// TIA Portal V20 export
DATA_BLOCK "DB_Digital_Outputs"   // DB3
{ S7_Optimized_Access := 'TRUE' }
// stored: MemoryReserve 100
   VAR
      Digital_Output_0 : Bool;
      Digital_Output_1 : Bool;
      Digital_Output_2 : Bool;
      Digital_Output_3 : Bool;
      Digital_Output_4 : Bool;
      Digital_Output_5 : Bool;
      Digital_Output_6 : Bool;
      Digital_Output_7 : Bool;
      Digital_Output_8 : Bool;
      Digital_Output_9 : Bool;
   END_VAR
BEGIN
END_DATA_BLOCK
